{attribute 'qualified_only'}
VAR_GLOBAL PERSISTENT
	rIntegratorResult:LREAL;
END_VAR

(* stored: Version 1.1.0.1, ProductVersion 3.1.4024.12
   GVL GVL_Math: Id {315a9746-0608-4a6b-94a6-cedf34feb45f} *)
